_CFC_ (* Continuous Function Chart, elements in execution order *)
#0 AND(SCHU_P2_3_Z_M1_AV, SCHU_P2_3_Z_M2_AV)
#1 OR(#0, #3)
#2 TON_OTK_MV:TON(IN: #1, PT: t#5s)
#3 AND(NOT SCHU_P2_3_SA1_DI5_A, NOT SCHU_P2_3_SA8_DI3_A, NOT SCHU_P2_3_SA1_DI6_M, NOT SCHU_P2_3_SA8_DI4_M)
#4 RT_Pusk:R_TRIG(CLK: SCHU_P2_3_UST_RE_PUSK)
#5 TON_PCH_OTKL:TON(IN: SCHU_P2_3_UST_RE_STOP, PT: T#1s)
#6 FT_PCH_OTKL:R_TRIG(CLK: #5.Q)
#7 RS_YA1_Open:RS(SET: #4.Q, RESET1: #6.Q)
#8 ZADERJ_SHOD_YA1:TON(IN: #7.Q1, PT: t#10s)
#9 TON_YA1_Z_ZAM_TE2:TON(IN: SCHU_P2_3_TE2_M_ZASCH, PT: t#5s)
#10 OR(#9.Q, Z_ZAM_SR, #2.Q)
#11 SEL(SCHU_P2_3_SA7_DI1_A, eHVAC2PointActuatorMode_Close_OP, eHVAC2PointActuatorMode_Auto_BMS)
#12 SEL(#10, #11, eHVAC2PointActuatorMode_Close_OP)
#13 fb_HVACPA:FB_HVAC2PointActuator(eHVACDataSecurityType_Idle, FALSE, TRUE, #8.Q, #12, SCHU_P2_3_KV1_DI4, SCHU_P2_3_YA1_DI6_ZKR, SCHU_P2_3_YA1_DI7_OTK, TRUE, SCHU_P2_3_SB, enableLimitSwitch, stokeTime)
#14 SCHU_P2_3_SA7_DO7_OTK <= #13.out 1
#15 OR(#13.out 4, #13.out 5)
#16 YA1_OTKAZ <= #15
#17 INT_TO_TIME(SCHU_P2_3_YA1_VREMYA_HODA)
#18 MUL(#17, 1000)
#19 stokeTime <= #18
_END_CFC_
END_PROGRAM
